PROGRAM MAIN
VAR
	wing : BOOL;
	cash : BOOL;
END_VAR

wing := cash;

END_PROGRAM

(* stored: Version 1.1.0.1, ProductVersion 3.1.4024.12
   POU MAIN: Id {fb865085-101d-43b2-9288-aeafc8caefc8}, SpecialFunc None *)
